Fanuc KAREL source: kd00020.KL

-- PROVISIONAL review KL for V770-1; original PC SHA256 18dfe7bef03fb2186dd76ff41ec21fe3b93e3fb32db646f2d9d4b45a5e52c383
-- Incomplete behavior may be omitted. Consult companion uncertainty JSON. Do not deploy.
PROGRAM KD00020
%NOLOCKGROUP
VAR
  I : INTEGER
  J : INTEGER
  B : BOOLEAN
  R : REAL
  S : STRING[80]
BEGIN
  -- UNRESOLVED_PC offsets 5-10; opcodes 7A
  -- UNRESOLVED_PC offsets 15-22; opcodes 9D,23
  -- UNRESOLVED_PC offsets 27-31; opcodes 7F
END KD00020
